Fanuc KAREL source: kt00333.KL

-- PROVISIONAL review KL for V940-1; original PC SHA256 adb0d5430db07c338bcb00e5514f17264d83bbdc02c40bcb7bda12ee582d71ed
-- Incomplete behavior may be omitted. Consult companion uncertainty JSON. Do not deploy.
PROGRAM KT00333
%NOLOCKGROUP
VAR
  R1 : REAL
  I2 : INTEGER
  OUT : BOOLEAN
BEGIN
  -- V9_ZERO_TABLE_METADATA_HINT layout=0001; no indexed target words; source/name/runtime held
  -- UNRESOLVED_PC offsets 5-16; opcodes 2E,23
  -- UNRESOLVED_PC offsets 21-32; opcodes 2E,23
  -- UNRESOLVED_PC offsets 37-57; opcodes 21,21,64,6F,23
  -- UNRESOLVED_PC offsets 62-66; opcodes 7F
END KT00333
